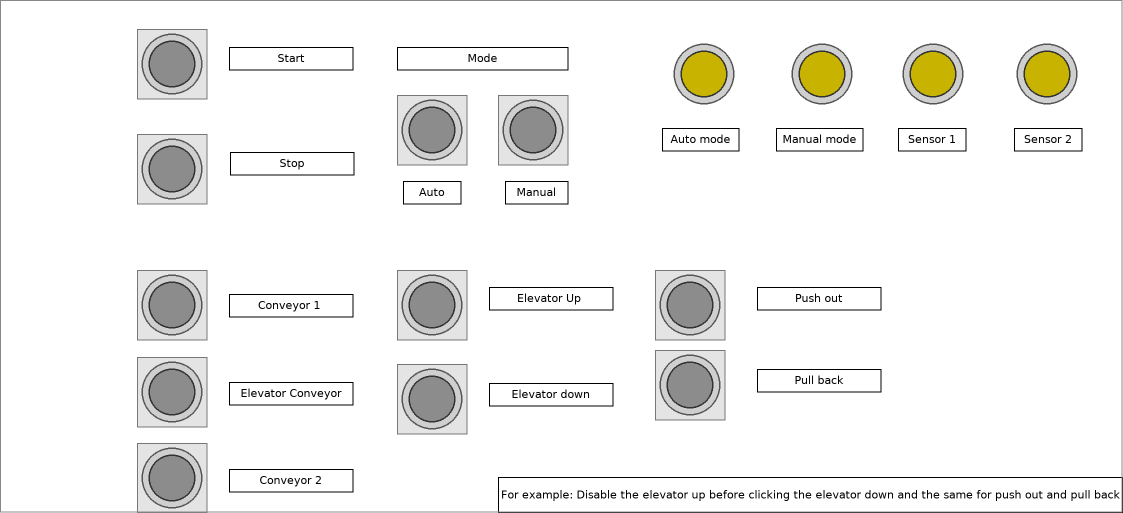
VISUALIZATION Visualization  // 1123x513
AR_IN_OUT
AR_IN_OUT
	
END_VAR
    PushSwitch (137,29 70x70), tooltip "START", variable: MAIN.START, behaviour: TOGGLE, style: Switch-PushSwitch-Gray
    PushSwitch (137,134 70x70), tooltip "Stop", variable: MAIN.STOP, behaviour: TOGGLE, style: Switch-PushSwitch-Gray
    PushSwitch (137,270 70x70), tooltip "Conv1", variable: MAIN.ManConveyor1, behaviour: TOGGLE, style: Switch-PushSwitch-Gray
    PushSwitch (137,443 70x70), tooltip "Conv2", variable: MAIN.ManConveyor2, behaviour: TOGGLE, style: Switch-PushSwitch-Gray
    PushSwitch (397,270 70x70), tooltip "up", variable: MAIN.ManElevatorUp, behaviour: TOGGLE, style: Switch-PushSwitch-Gray
    PushSwitch (397,364 70x70), tooltip "down", variable: MAIN.ManElevatorDown, behaviour: TOGGLE, style: Switch-PushSwitch-Gray
    PushSwitch (655,270 70x70), tooltip "push", variable: MAIN.ManPusherPush, behaviour: TOGGLE, style: Switch-PushSwitch-Gray
    PushSwitch (655,350 70x70), tooltip "retract", variable: MAIN.ManPusherRetract, behaviour: TOGGLE, style: Switch-PushSwitch-Gray
    PushSwitch (397,95 70x70), tooltip "Auto_mode", variable: MAIN.Auto_mode, behaviour: TOGGLE, style: Switch-PushSwitch-Gray
    PushSwitch (498,95 70x70), tooltip "Manual mode", variable: MAIN.Manual_mode, behaviour: TOGGLE, style: Switch-PushSwitch-Gray
    PushSwitch (137,357 70x70), tooltip "Conv1", variable: MAIN.ManElevatorConveyor, behaviour: TOGGLE, style: Switch-PushSwitch-Gray
    Rectangle (397,47 171x23), "Mode"
    Rectangle (403,181 58x23), "Auto"
    Rectangle (505,181 63x23), "Manual"
    Rectangle (229,47 124x23), "Start"
    Rectangle (230,152 124x23), "Stop"
    Rectangle (229,294 124x23), "Conveyor 1"
    Rectangle (229,382 124x23), "Elevator Conveyor"
    Rectangle (489,287 124x23), "Elevator Up"
    Rectangle (489,383 124x23), "Elevator down"
    Rectangle (229,469 124x23), "Conveyor 2"
    Rectangle (757,287 124x23), "Push out"
    Rectangle (757,369 124x23), "Pull back"
    Lamp1 (1012,39 70x70), variable: MAIN.iConveyor2Sensor, style: Lamp-Lamp1-Yellow
    Lamp1 (898,39 70x70), variable: MAIN.iElevatorSensor, style: Lamp-Lamp1-Yellow
    Rectangle (898,128 68x23), "Sensor 1"
    Rectangle (1014,128 68x23), "Sensor 2"
    Lamp1 (669,39 70x70), variable: MAIN.Auto_mode, style: Lamp-Lamp1-Yellow
    Lamp1 (787,39 70x70), variable: MAIN.Manual_mode, style: Lamp-Lamp1-Yellow
    Rectangle (662,128 77x23), "Auto mode"
    Rectangle (776,128 87x23), "Manual mode"
    Rectangle (498,477 625x36), "For example: Disable the elevator up before clicking the elevator down and the same for push out and pull back"
END_VISUALIZATION

(* stored: Version 1.1.0.1
   Visu Visualization: Id {ce8fd711-03f3-42e0-875b-89585811f50a} *)
